// TIA Portal V15.1 export
// export: Created 2026-01-09T13:45:15.2149014Z, ExportSetting WithDefaults, WithReadOnly, DisplayName Totally Integrated Automation Portal, DisplayVersion V15.1 Update 8, DisplayName TIA Portal Openness, DisplayVersion V15.1 Update 8, DisplayName STEP 7 Professional, DisplayVersion V15.1 Update 8, DisplayName WinCC Advanced, DisplayVersion V15.1 Update 8
FUNCTION "FCCA_CCD_AGG12345" : Void   // FC19, LAD
{ S7_Optimized_Access := 'TRUE' }
VERSION : 0.1
// stored: AutoNumber true, CodeModifiedDate 2026-01-04T14:27:04.5188811Z, CompileDate 2026-01-04T14:27:06.4720109Z, CreationDate 2024-10-13T15:07:34.9617085Z, HandleErrorsWithinBlock false, InterfaceModifiedDate 2024-08-08T03:15:59.3806622Z, IsConsistent true, IsIECCheckEnabled false, IsKnowHowProtected false, IsWriteProtected false, LibraryConformanceStatus Error: The block contains calls of single instances. Warning: The object contains access to global data blocks. Warning: The block contains direct access to inputs, outputs, bit memories, indirect access to the registry or indirect access to external memory areas that are unknown at the time of compilation., ModifiedDate 2026-01-04T14:27:04.5188811Z, ParameterModified 2024-08-08T03:15:59.3806622Z, PLCSimAdvancedSupport false, SetENOAutomatically False, StructureModified 2024-08-08T03:15:59.3806622Z, UDAEnableTagReadback false
   VAR_TEMP   // added for the SCL form of the ladder/FBD networks
      _w1 : Bool;
   END_VAR
BEGIN

REGION Network 1: CAN COT LIEU AGG1
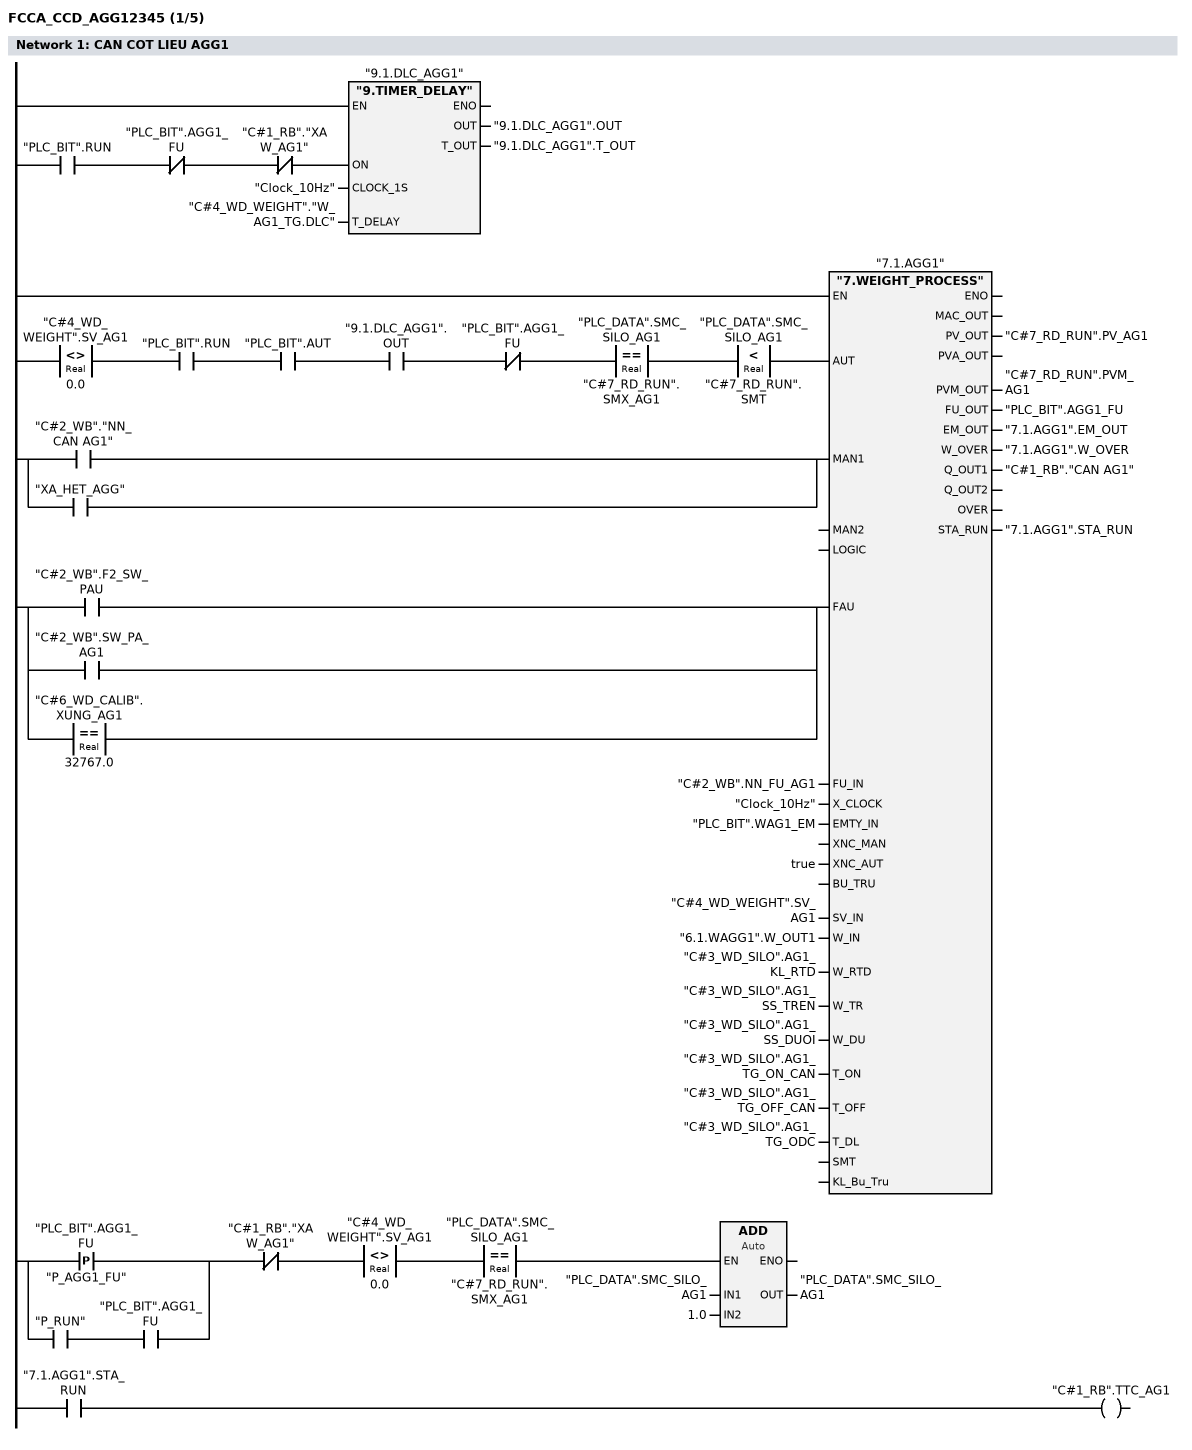
   RUNG wire#powerrail
      "9.1.DLC_AGG1"(ON := wire#w1, CLOCK_1S := "Clock_10Hz", T_DELAY := "C#4_WD_WEIGHT"."W_AG1_TG.DLC", OUT => "9.1.DLC_AGG1".OUT, T_OUT => "9.1.DLC_AGG1".T_OUT)
   END_RUNG
   RUNG wire#powerrail
      Contact( "PLC_BIT".RUN )
      I_Contact( "PLC_BIT".AGG1_FU )
      I_Contact( "C#1_RB"."XA W_AG1" )
   END_RUNG wire#w1
   RUNG wire#powerrail
      "7.1.AGG1"(AUT := wire#w2, MAN1 := wire#w3, FAU := wire#w4, MAN2 :=, LOGIC :=, FU_IN := "C#2_WB".NN_FU_AG1, X_CLOCK := "Clock_10Hz", EMTY_IN := "PLC_BIT".WAG1_EM, XNC_MAN :=, XNC_AUT := true, BU_TRU :=, SV_IN := "C#4_WD_WEIGHT".SV_AG1, W_IN := "6.1.WAGG1".W_OUT1, W_RTD := "C#3_WD_SILO".AG1_KL_RTD, W_TR := "C#3_WD_SILO".AG1_SS_TREN, W_DU := "C#3_WD_SILO".AG1_SS_DUOI, T_ON := "C#3_WD_SILO".AG1_TG_ON_CAN, T_OFF := "C#3_WD_SILO".AG1_TG_OFF_CAN, T_DL := "C#3_WD_SILO".AG1_TG_ODC, SMT :=, KL_Bu_Tru :=, MAC_OUT =>, PV_OUT => "C#7_RD_RUN".PV_AG1, PVA_OUT =>, PVM_OUT => "C#7_RD_RUN".PVM_AG1, FU_OUT => "PLC_BIT".AGG1_FU, EM_OUT => "7.1.AGG1".EM_OUT, W_OVER => "7.1.AGG1".W_OVER, Q_OUT1 => "C#1_RB"."CAN AG1", Q_OUT2 =>, OVER =>, STA_RUN => "7.1.AGG1".STA_RUN)
   END_RUNG
   RUNG wire#powerrail
      { S7_Templates := "SrcType := Real" } NE_Contact(in1 := "C#4_WD_WEIGHT".SV_AG1, in2 := 0.0)
      Contact( "PLC_BIT".RUN )
      Contact( "PLC_BIT".AUT )
      Contact( "9.1.DLC_AGG1".OUT )
      I_Contact( "PLC_BIT".AGG1_FU )
      { S7_Templates := "SrcType := Real" } EQ_Contact(in1 := "PLC_DATA".SMC_SILO_AG1, in2 := "C#7_RD_RUN".SMX_AG1)
      { S7_Templates := "SrcType := Real" } LT_Contact(in1 := "PLC_DATA".SMC_SILO_AG1, in2 := "C#7_RD_RUN".SMT)
   END_RUNG wire#w2
   RUNG wire#powerrail
      Contact( "C#2_WB"."NN_CAN AG1" )
   END_RUNG wire#w3
   RUNG wire#powerrail
      Contact( "XA_HET_AGG" )
   END_RUNG wire#w3
   RUNG wire#powerrail
      Contact( "C#2_WB".F2_SW_PAU )
   END_RUNG wire#w4
   RUNG wire#powerrail
      Contact( "C#2_WB".SW_PA_AG1 )
   END_RUNG wire#w4
   RUNG wire#powerrail
      { S7_Templates := "SrcType := Real" } EQ_Contact(in1 := "C#6_WD_CALIB".XUNG_AG1, in2 := 32767.0)
   END_RUNG wire#w4
   RUNG wire#powerrail
      P_Contact(operand := "PLC_BIT".AGG1_FU, bit := "P_AGG1_FU")
      wire#w5
      I_Contact( "C#1_RB"."XA W_AG1" )
      { S7_Templates := "SrcType := Real" } NE_Contact(in1 := "C#4_WD_WEIGHT".SV_AG1, in2 := 0.0)
      { S7_Templates := "SrcType := Real" } EQ_Contact(in1 := "PLC_DATA".SMC_SILO_AG1, in2 := "C#7_RD_RUN".SMX_AG1)
      Add(in1 := "PLC_DATA".SMC_SILO_AG1, in2 := 1.0, out => "PLC_DATA".SMC_SILO_AG1)
   END_RUNG
   RUNG wire#powerrail
      Contact( "P_RUN" )
      Contact( "PLC_BIT".AGG1_FU )
   END_RUNG wire#w5
   RUNG wire#powerrail
      Contact( "7.1.AGG1".STA_RUN )
      Coil( "C#1_RB".TTC_AG1 )
   END_RUNG
   // the same network as SCL:
   "9.1.DLC_AGG1"(ON := "PLC_BIT".RUN AND NOT "PLC_BIT".AGG1_FU AND NOT "C#1_RB"."XA W_AG1",   // "9.TIMER_DELAY"
                  CLOCK_1S := "Clock_10Hz",
                  T_DELAY := "C#4_WD_WEIGHT"."W_AG1_TG.DLC",
                  OUT => "9.1.DLC_AGG1".OUT,
                  T_OUT => "9.1.DLC_AGG1".T_OUT);
   "7.1.AGG1"(AUT := ("C#4_WD_WEIGHT".SV_AG1 <> 0.0) AND "PLC_BIT".RUN AND "PLC_BIT".AUT AND "9.1.DLC_AGG1".OUT AND NOT "PLC_BIT".AGG1_FU AND ("PLC_DATA".SMC_SILO_AG1 = "C#7_RD_RUN".SMX_AG1) AND ("PLC_DATA".SMC_SILO_AG1 < "C#7_RD_RUN".SMT),   // "7.WEIGHT_PROCESS"
              MAN1 := "C#2_WB"."NN_CAN AG1" OR "XA_HET_AGG",
              FAU := "C#2_WB".F2_SW_PAU OR "C#2_WB".SW_PA_AG1 OR ("C#6_WD_CALIB".XUNG_AG1 = 32767.0),
              FU_IN := "C#2_WB".NN_FU_AG1,
              X_CLOCK := "Clock_10Hz",
              EMTY_IN := "PLC_BIT".WAG1_EM,
              XNC_AUT := true,
              SV_IN := "C#4_WD_WEIGHT".SV_AG1,
              W_IN := "6.1.WAGG1".W_OUT1,
              W_RTD := "C#3_WD_SILO".AG1_KL_RTD,
              W_TR := "C#3_WD_SILO".AG1_SS_TREN,
              W_DU := "C#3_WD_SILO".AG1_SS_DUOI,
              T_ON := "C#3_WD_SILO".AG1_TG_ON_CAN,
              T_OFF := "C#3_WD_SILO".AG1_TG_OFF_CAN,
              T_DL := "C#3_WD_SILO".AG1_TG_ODC,
              PV_OUT => "C#7_RD_RUN".PV_AG1,
              PVM_OUT => "C#7_RD_RUN".PVM_AG1,
              FU_OUT => "PLC_BIT".AGG1_FU,
              EM_OUT => "7.1.AGG1".EM_OUT,
              W_OVER => "7.1.AGG1".W_OVER,
              Q_OUT1 => "C#1_RB"."CAN AG1",
              STA_RUN => "7.1.AGG1".STA_RUN);
   #_w1 := "PLC_BIT".AGG1_FU AND NOT "P_AGG1_FU";   // rising edge of "PLC_BIT".AGG1_FU
   "P_AGG1_FU" := "PLC_BIT".AGG1_FU;
   IF (#_w1 OR ("P_RUN" AND "PLC_BIT".AGG1_FU)) AND NOT "C#1_RB"."XA W_AG1" AND ("C#4_WD_WEIGHT".SV_AG1 <> 0.0) AND ("PLC_DATA".SMC_SILO_AG1 = "C#7_RD_RUN".SMX_AG1) THEN
       "PLC_DATA".SMC_SILO_AG1 := "PLC_DATA".SMC_SILO_AG1 + 1.0;
   END_IF;
   "C#1_RB".TTC_AG1 := "7.1.AGG1".STA_RUN;
END_REGION

REGION Network 2: CAN COT LIEU AGG2
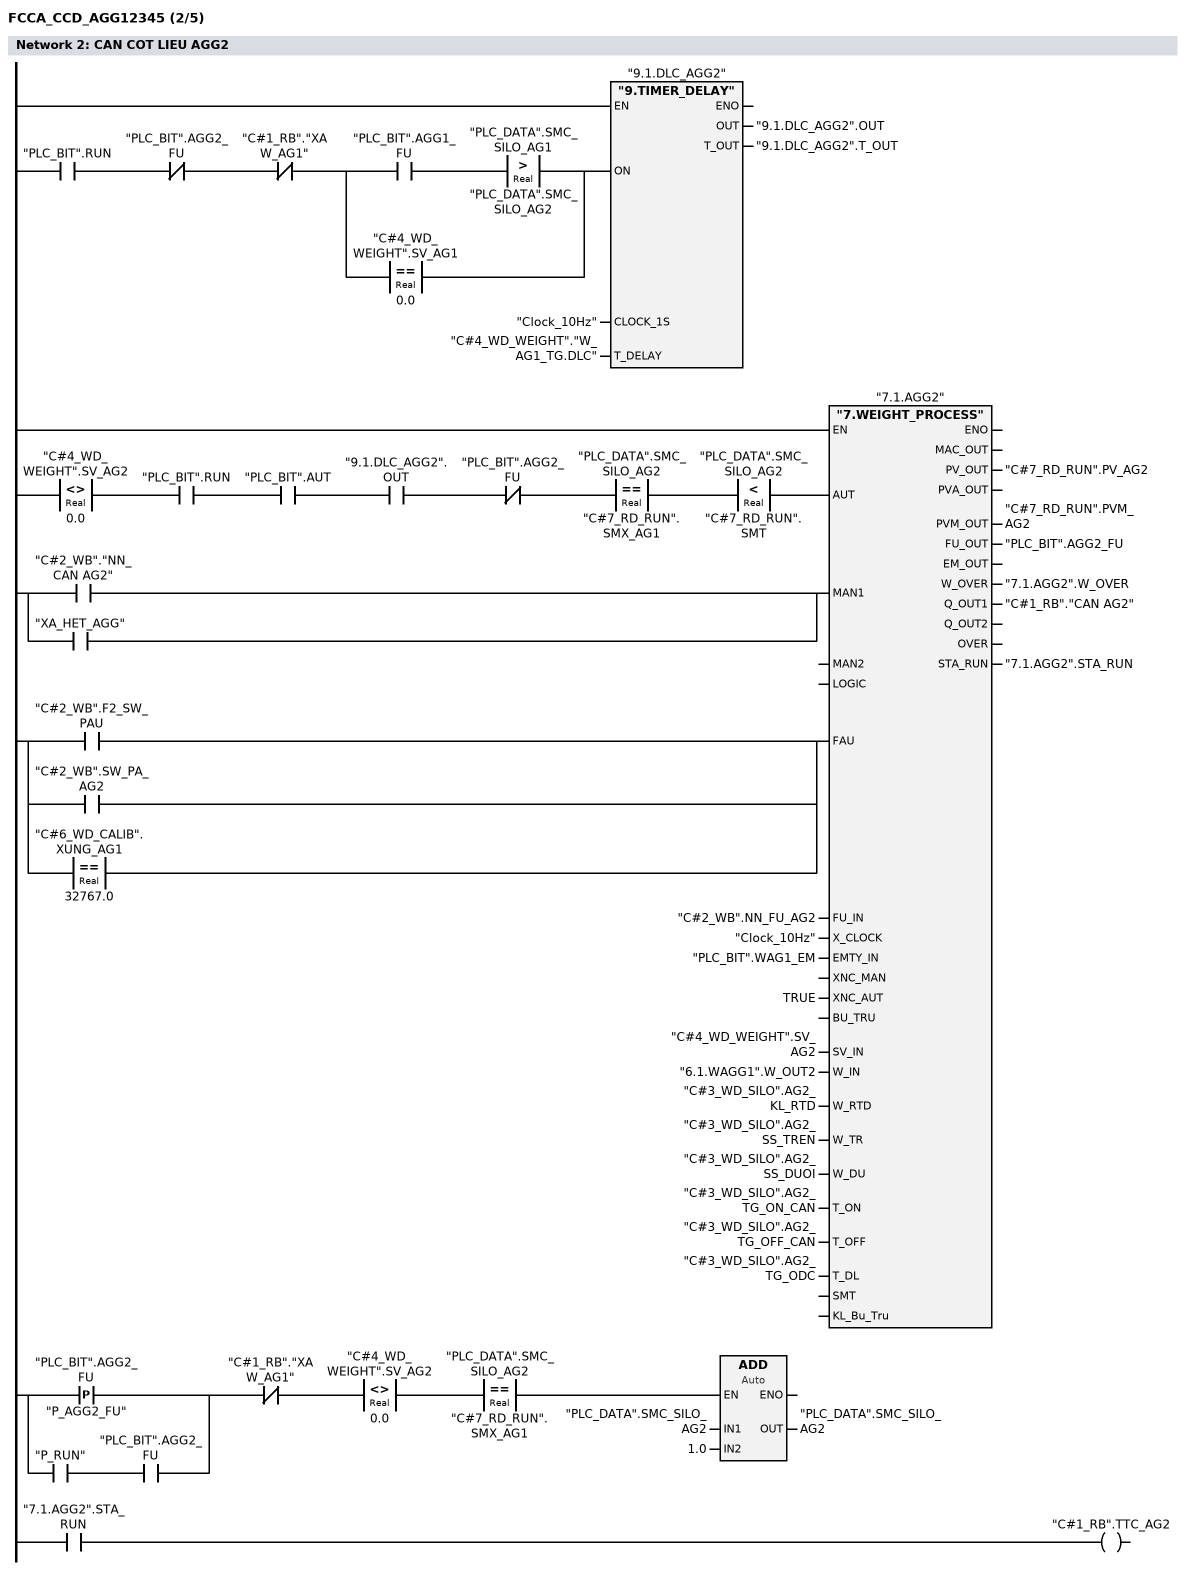
   RUNG wire#powerrail
      "9.1.DLC_AGG2"(ON := wire#w2, CLOCK_1S := "Clock_10Hz", T_DELAY := "C#4_WD_WEIGHT"."W_AG1_TG.DLC", OUT => "9.1.DLC_AGG2".OUT, T_OUT => "9.1.DLC_AGG2".T_OUT)
   END_RUNG
   RUNG wire#powerrail
      Contact( "PLC_BIT".RUN )
      I_Contact( "PLC_BIT".AGG2_FU )
      I_Contact( "C#1_RB"."XA W_AG1" )
      wire#w1
      Contact( "PLC_BIT".AGG1_FU )
      { S7_Templates := "SrcType := Real" } GT_Contact(in1 := "PLC_DATA".SMC_SILO_AG1, in2 := "PLC_DATA".SMC_SILO_AG2)
   END_RUNG wire#w2
   RUNG wire#w1
      { S7_Templates := "SrcType := Real" } EQ_Contact(in1 := "C#4_WD_WEIGHT".SV_AG1, in2 := 0.0)
   END_RUNG wire#w2
   RUNG wire#powerrail
      "7.1.AGG2"(AUT := wire#w3, MAN1 := wire#w4, FAU := wire#w5, MAN2 :=, LOGIC :=, FU_IN := "C#2_WB".NN_FU_AG2, X_CLOCK := "Clock_10Hz", EMTY_IN := "PLC_BIT".WAG1_EM, XNC_MAN :=, XNC_AUT := TRUE, BU_TRU :=, SV_IN := "C#4_WD_WEIGHT".SV_AG2, W_IN := "6.1.WAGG1".W_OUT2, W_RTD := "C#3_WD_SILO".AG2_KL_RTD, W_TR := "C#3_WD_SILO".AG2_SS_TREN, W_DU := "C#3_WD_SILO".AG2_SS_DUOI, T_ON := "C#3_WD_SILO".AG2_TG_ON_CAN, T_OFF := "C#3_WD_SILO".AG2_TG_OFF_CAN, T_DL := "C#3_WD_SILO".AG2_TG_ODC, SMT :=, KL_Bu_Tru :=, MAC_OUT =>, PV_OUT => "C#7_RD_RUN".PV_AG2, PVA_OUT =>, PVM_OUT => "C#7_RD_RUN".PVM_AG2, FU_OUT => "PLC_BIT".AGG2_FU, EM_OUT =>, W_OVER => "7.1.AGG2".W_OVER, Q_OUT1 => "C#1_RB"."CAN AG2", Q_OUT2 =>, OVER =>, STA_RUN => "7.1.AGG2".STA_RUN)
   END_RUNG
   RUNG wire#powerrail
      { S7_Templates := "SrcType := Real" } NE_Contact(in1 := "C#4_WD_WEIGHT".SV_AG2, in2 := 0.0)
      Contact( "PLC_BIT".RUN )
      Contact( "PLC_BIT".AUT )
      Contact( "9.1.DLC_AGG2".OUT )
      I_Contact( "PLC_BIT".AGG2_FU )
      { S7_Templates := "SrcType := Real" } EQ_Contact(in1 := "PLC_DATA".SMC_SILO_AG2, in2 := "C#7_RD_RUN".SMX_AG1)
      { S7_Templates := "SrcType := Real" } LT_Contact(in1 := "PLC_DATA".SMC_SILO_AG2, in2 := "C#7_RD_RUN".SMT)
   END_RUNG wire#w3
   RUNG wire#powerrail
      Contact( "C#2_WB"."NN_CAN AG2" )
   END_RUNG wire#w4
   RUNG wire#powerrail
      Contact( "XA_HET_AGG" )
   END_RUNG wire#w4
   RUNG wire#powerrail
      Contact( "C#2_WB".F2_SW_PAU )
   END_RUNG wire#w5
   RUNG wire#powerrail
      Contact( "C#2_WB".SW_PA_AG2 )
   END_RUNG wire#w5
   RUNG wire#powerrail
      { S7_Templates := "SrcType := Real" } EQ_Contact(in1 := "C#6_WD_CALIB".XUNG_AG1, in2 := 32767.0)
   END_RUNG wire#w5
   RUNG wire#powerrail
      P_Contact(operand := "PLC_BIT".AGG2_FU, bit := "P_AGG2_FU")
      wire#w6
      I_Contact( "C#1_RB"."XA W_AG1" )
      { S7_Templates := "SrcType := Real" } NE_Contact(in1 := "C#4_WD_WEIGHT".SV_AG2, in2 := 0.0)
      { S7_Templates := "SrcType := Real" } EQ_Contact(in1 := "PLC_DATA".SMC_SILO_AG2, in2 := "C#7_RD_RUN".SMX_AG1)
      Add(in1 := "PLC_DATA".SMC_SILO_AG2, in2 := 1.0, out => "PLC_DATA".SMC_SILO_AG2)
   END_RUNG
   RUNG wire#powerrail
      Contact( "P_RUN" )
      Contact( "PLC_BIT".AGG2_FU )
   END_RUNG wire#w6
   RUNG wire#powerrail
      Contact( "7.1.AGG2".STA_RUN )
      Coil( "C#1_RB".TTC_AG2 )
   END_RUNG
   // the same network as SCL:
   "9.1.DLC_AGG2"(ON := "PLC_BIT".RUN AND NOT "PLC_BIT".AGG2_FU AND NOT "C#1_RB"."XA W_AG1" AND (("PLC_BIT".AGG1_FU AND ("PLC_DATA".SMC_SILO_AG1 > "PLC_DATA".SMC_SILO_AG2)) OR ("C#4_WD_WEIGHT".SV_AG1 = 0.0)),   // "9.TIMER_DELAY"
                  CLOCK_1S := "Clock_10Hz",
                  T_DELAY := "C#4_WD_WEIGHT"."W_AG1_TG.DLC",
                  OUT => "9.1.DLC_AGG2".OUT,
                  T_OUT => "9.1.DLC_AGG2".T_OUT);
   "7.1.AGG2"(AUT := ("C#4_WD_WEIGHT".SV_AG2 <> 0.0) AND "PLC_BIT".RUN AND "PLC_BIT".AUT AND "9.1.DLC_AGG2".OUT AND NOT "PLC_BIT".AGG2_FU AND ("PLC_DATA".SMC_SILO_AG2 = "C#7_RD_RUN".SMX_AG1) AND ("PLC_DATA".SMC_SILO_AG2 < "C#7_RD_RUN".SMT),   // "7.WEIGHT_PROCESS"
              MAN1 := "C#2_WB"."NN_CAN AG2" OR "XA_HET_AGG",
              FAU := "C#2_WB".F2_SW_PAU OR "C#2_WB".SW_PA_AG2 OR ("C#6_WD_CALIB".XUNG_AG1 = 32767.0),
              FU_IN := "C#2_WB".NN_FU_AG2,
              X_CLOCK := "Clock_10Hz",
              EMTY_IN := "PLC_BIT".WAG1_EM,
              XNC_AUT := TRUE,
              SV_IN := "C#4_WD_WEIGHT".SV_AG2,
              W_IN := "6.1.WAGG1".W_OUT2,
              W_RTD := "C#3_WD_SILO".AG2_KL_RTD,
              W_TR := "C#3_WD_SILO".AG2_SS_TREN,
              W_DU := "C#3_WD_SILO".AG2_SS_DUOI,
              T_ON := "C#3_WD_SILO".AG2_TG_ON_CAN,
              T_OFF := "C#3_WD_SILO".AG2_TG_OFF_CAN,
              T_DL := "C#3_WD_SILO".AG2_TG_ODC,
              PV_OUT => "C#7_RD_RUN".PV_AG2,
              PVM_OUT => "C#7_RD_RUN".PVM_AG2,
              FU_OUT => "PLC_BIT".AGG2_FU,
              W_OVER => "7.1.AGG2".W_OVER,
              Q_OUT1 => "C#1_RB"."CAN AG2",
              STA_RUN => "7.1.AGG2".STA_RUN);
   #_w1 := "PLC_BIT".AGG2_FU AND NOT "P_AGG2_FU";   // rising edge of "PLC_BIT".AGG2_FU
   "P_AGG2_FU" := "PLC_BIT".AGG2_FU;
   IF (#_w1 OR ("P_RUN" AND "PLC_BIT".AGG2_FU)) AND NOT "C#1_RB"."XA W_AG1" AND ("C#4_WD_WEIGHT".SV_AG2 <> 0.0) AND ("PLC_DATA".SMC_SILO_AG2 = "C#7_RD_RUN".SMX_AG1) THEN
       "PLC_DATA".SMC_SILO_AG2 := "PLC_DATA".SMC_SILO_AG2 + 1.0;
   END_IF;
   "C#1_RB".TTC_AG2 := "7.1.AGG2".STA_RUN;
END_REGION

REGION Network 3: CAN COT LIEU AGG3
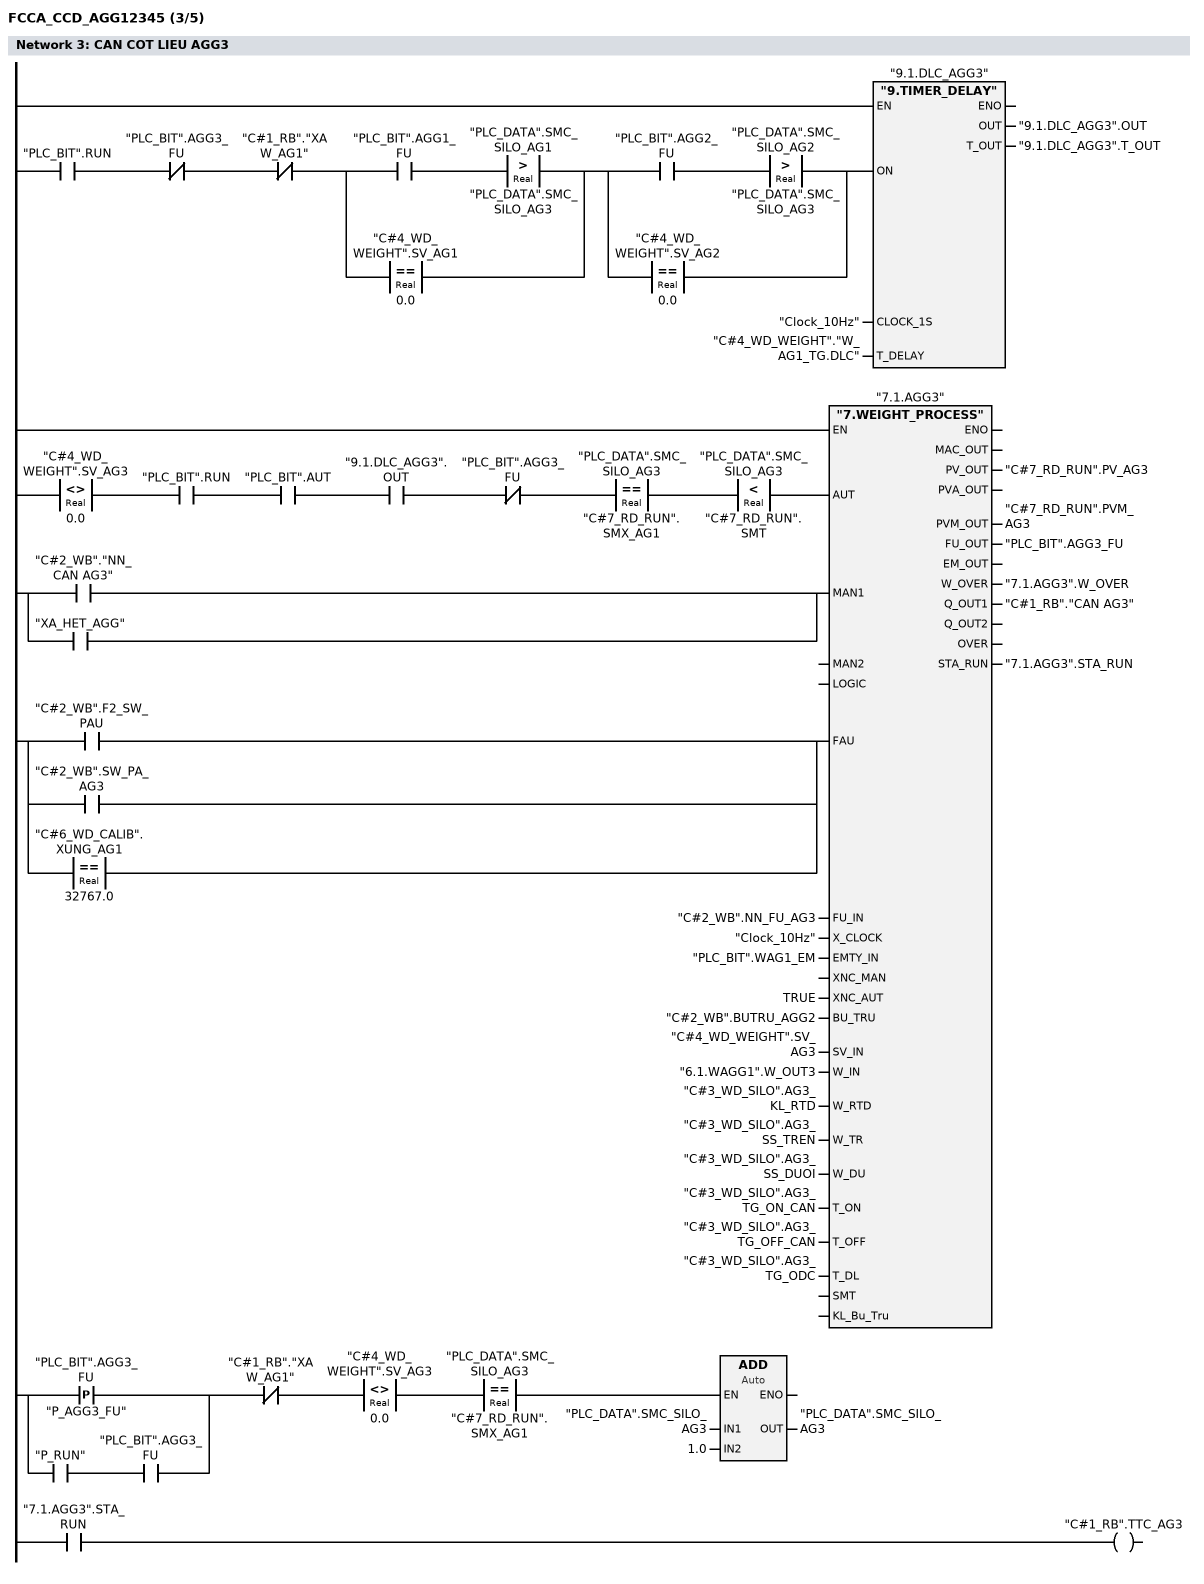
   RUNG wire#powerrail
      "9.1.DLC_AGG3"(ON := wire#w3, CLOCK_1S := "Clock_10Hz", T_DELAY := "C#4_WD_WEIGHT"."W_AG1_TG.DLC", OUT => "9.1.DLC_AGG3".OUT, T_OUT => "9.1.DLC_AGG3".T_OUT)
   END_RUNG
   RUNG wire#powerrail
      Contact( "PLC_BIT".RUN )
      I_Contact( "PLC_BIT".AGG3_FU )
      I_Contact( "C#1_RB"."XA W_AG1" )
      wire#w1
      Contact( "PLC_BIT".AGG1_FU )
      { S7_Templates := "SrcType := Real" } GT_Contact(in1 := "PLC_DATA".SMC_SILO_AG1, in2 := "PLC_DATA".SMC_SILO_AG3)
      wire#w2
      Contact( "PLC_BIT".AGG2_FU )
      { S7_Templates := "SrcType := Real" } GT_Contact(in1 := "PLC_DATA".SMC_SILO_AG2, in2 := "PLC_DATA".SMC_SILO_AG3)
   END_RUNG wire#w3
   RUNG wire#w1
      { S7_Templates := "SrcType := Real" } EQ_Contact(in1 := "C#4_WD_WEIGHT".SV_AG1, in2 := 0.0)
   END_RUNG wire#w2
   RUNG wire#w2
      { S7_Templates := "SrcType := Real" } EQ_Contact(in1 := "C#4_WD_WEIGHT".SV_AG2, in2 := 0.0)
   END_RUNG wire#w3
   RUNG wire#powerrail
      "7.1.AGG3"(AUT := wire#w4, MAN1 := wire#w5, FAU := wire#w6, MAN2 :=, LOGIC :=, FU_IN := "C#2_WB".NN_FU_AG3, X_CLOCK := "Clock_10Hz", EMTY_IN := "PLC_BIT".WAG1_EM, XNC_MAN :=, XNC_AUT := TRUE, BU_TRU := "C#2_WB".BUTRU_AGG2, SV_IN := "C#4_WD_WEIGHT".SV_AG3, W_IN := "6.1.WAGG1".W_OUT3, W_RTD := "C#3_WD_SILO".AG3_KL_RTD, W_TR := "C#3_WD_SILO".AG3_SS_TREN, W_DU := "C#3_WD_SILO".AG3_SS_DUOI, T_ON := "C#3_WD_SILO".AG3_TG_ON_CAN, T_OFF := "C#3_WD_SILO".AG3_TG_OFF_CAN, T_DL := "C#3_WD_SILO".AG3_TG_ODC, SMT :=, KL_Bu_Tru :=, MAC_OUT =>, PV_OUT => "C#7_RD_RUN".PV_AG3, PVA_OUT =>, PVM_OUT => "C#7_RD_RUN".PVM_AG3, FU_OUT => "PLC_BIT".AGG3_FU, EM_OUT =>, W_OVER => "7.1.AGG3".W_OVER, Q_OUT1 => "C#1_RB"."CAN AG3", Q_OUT2 =>, OVER =>, STA_RUN => "7.1.AGG3".STA_RUN)
   END_RUNG
   RUNG wire#powerrail
      { S7_Templates := "SrcType := Real" } NE_Contact(in1 := "C#4_WD_WEIGHT".SV_AG3, in2 := 0.0)
      Contact( "PLC_BIT".RUN )
      Contact( "PLC_BIT".AUT )
      Contact( "9.1.DLC_AGG3".OUT )
      I_Contact( "PLC_BIT".AGG3_FU )
      { S7_Templates := "SrcType := Real" } EQ_Contact(in1 := "PLC_DATA".SMC_SILO_AG3, in2 := "C#7_RD_RUN".SMX_AG1)
      { S7_Templates := "SrcType := Real" } LT_Contact(in1 := "PLC_DATA".SMC_SILO_AG3, in2 := "C#7_RD_RUN".SMT)
   END_RUNG wire#w4
   RUNG wire#powerrail
      Contact( "C#2_WB"."NN_CAN AG3" )
   END_RUNG wire#w5
   RUNG wire#powerrail
      Contact( "XA_HET_AGG" )
   END_RUNG wire#w5
   RUNG wire#powerrail
      Contact( "C#2_WB".F2_SW_PAU )
   END_RUNG wire#w6
   RUNG wire#powerrail
      Contact( "C#2_WB".SW_PA_AG3 )
   END_RUNG wire#w6
   RUNG wire#powerrail
      { S7_Templates := "SrcType := Real" } EQ_Contact(in1 := "C#6_WD_CALIB".XUNG_AG1, in2 := 32767.0)
   END_RUNG wire#w6
   RUNG wire#powerrail
      P_Contact(operand := "PLC_BIT".AGG3_FU, bit := "P_AGG3_FU")
      wire#w7
      I_Contact( "C#1_RB"."XA W_AG1" )
      { S7_Templates := "SrcType := Real" } NE_Contact(in1 := "C#4_WD_WEIGHT".SV_AG3, in2 := 0.0)
      { S7_Templates := "SrcType := Real" } EQ_Contact(in1 := "PLC_DATA".SMC_SILO_AG3, in2 := "C#7_RD_RUN".SMX_AG1)
      Add(in1 := "PLC_DATA".SMC_SILO_AG3, in2 := 1.0, out => "PLC_DATA".SMC_SILO_AG3)
   END_RUNG
   RUNG wire#powerrail
      Contact( "P_RUN" )
      Contact( "PLC_BIT".AGG3_FU )
   END_RUNG wire#w7
   RUNG wire#powerrail
      Contact( "7.1.AGG3".STA_RUN )
      Coil( "C#1_RB".TTC_AG3 )
   END_RUNG
   // the same network as SCL:
   "9.1.DLC_AGG3"(ON := "PLC_BIT".RUN AND NOT "PLC_BIT".AGG3_FU AND NOT "C#1_RB"."XA W_AG1" AND (("PLC_BIT".AGG1_FU AND ("PLC_DATA".SMC_SILO_AG1 > "PLC_DATA".SMC_SILO_AG3)) OR ("C#4_WD_WEIGHT".SV_AG1 = 0.0)) AND (("PLC_BIT".AGG2_FU AND ("PLC_DATA".SMC_SILO_AG2 > "PLC_DATA".SMC_SILO_AG3)) OR ("C#4_WD_WEIGHT".SV_AG2 = 0.0)),   // "9.TIMER_DELAY"
                  CLOCK_1S := "Clock_10Hz",
                  T_DELAY := "C#4_WD_WEIGHT"."W_AG1_TG.DLC",
                  OUT => "9.1.DLC_AGG3".OUT,
                  T_OUT => "9.1.DLC_AGG3".T_OUT);
   "7.1.AGG3"(AUT := ("C#4_WD_WEIGHT".SV_AG3 <> 0.0) AND "PLC_BIT".RUN AND "PLC_BIT".AUT AND "9.1.DLC_AGG3".OUT AND NOT "PLC_BIT".AGG3_FU AND ("PLC_DATA".SMC_SILO_AG3 = "C#7_RD_RUN".SMX_AG1) AND ("PLC_DATA".SMC_SILO_AG3 < "C#7_RD_RUN".SMT),   // "7.WEIGHT_PROCESS"
              MAN1 := "C#2_WB"."NN_CAN AG3" OR "XA_HET_AGG",
              FAU := "C#2_WB".F2_SW_PAU OR "C#2_WB".SW_PA_AG3 OR ("C#6_WD_CALIB".XUNG_AG1 = 32767.0),
              FU_IN := "C#2_WB".NN_FU_AG3,
              X_CLOCK := "Clock_10Hz",
              EMTY_IN := "PLC_BIT".WAG1_EM,
              XNC_AUT := TRUE,
              BU_TRU := "C#2_WB".BUTRU_AGG2,
              SV_IN := "C#4_WD_WEIGHT".SV_AG3,
              W_IN := "6.1.WAGG1".W_OUT3,
              W_RTD := "C#3_WD_SILO".AG3_KL_RTD,
              W_TR := "C#3_WD_SILO".AG3_SS_TREN,
              W_DU := "C#3_WD_SILO".AG3_SS_DUOI,
              T_ON := "C#3_WD_SILO".AG3_TG_ON_CAN,
              T_OFF := "C#3_WD_SILO".AG3_TG_OFF_CAN,
              T_DL := "C#3_WD_SILO".AG3_TG_ODC,
              PV_OUT => "C#7_RD_RUN".PV_AG3,
              PVM_OUT => "C#7_RD_RUN".PVM_AG3,
              FU_OUT => "PLC_BIT".AGG3_FU,
              W_OVER => "7.1.AGG3".W_OVER,
              Q_OUT1 => "C#1_RB"."CAN AG3",
              STA_RUN => "7.1.AGG3".STA_RUN);
   #_w1 := "PLC_BIT".AGG3_FU AND NOT "P_AGG3_FU";   // rising edge of "PLC_BIT".AGG3_FU
   "P_AGG3_FU" := "PLC_BIT".AGG3_FU;
   IF (#_w1 OR ("P_RUN" AND "PLC_BIT".AGG3_FU)) AND NOT "C#1_RB"."XA W_AG1" AND ("C#4_WD_WEIGHT".SV_AG3 <> 0.0) AND ("PLC_DATA".SMC_SILO_AG3 = "C#7_RD_RUN".SMX_AG1) THEN
       "PLC_DATA".SMC_SILO_AG3 := "PLC_DATA".SMC_SILO_AG3 + 1.0;
   END_IF;
   "C#1_RB".TTC_AG3 := "7.1.AGG3".STA_RUN;
END_REGION

REGION Network 4: CAN COT LIEU AGG4
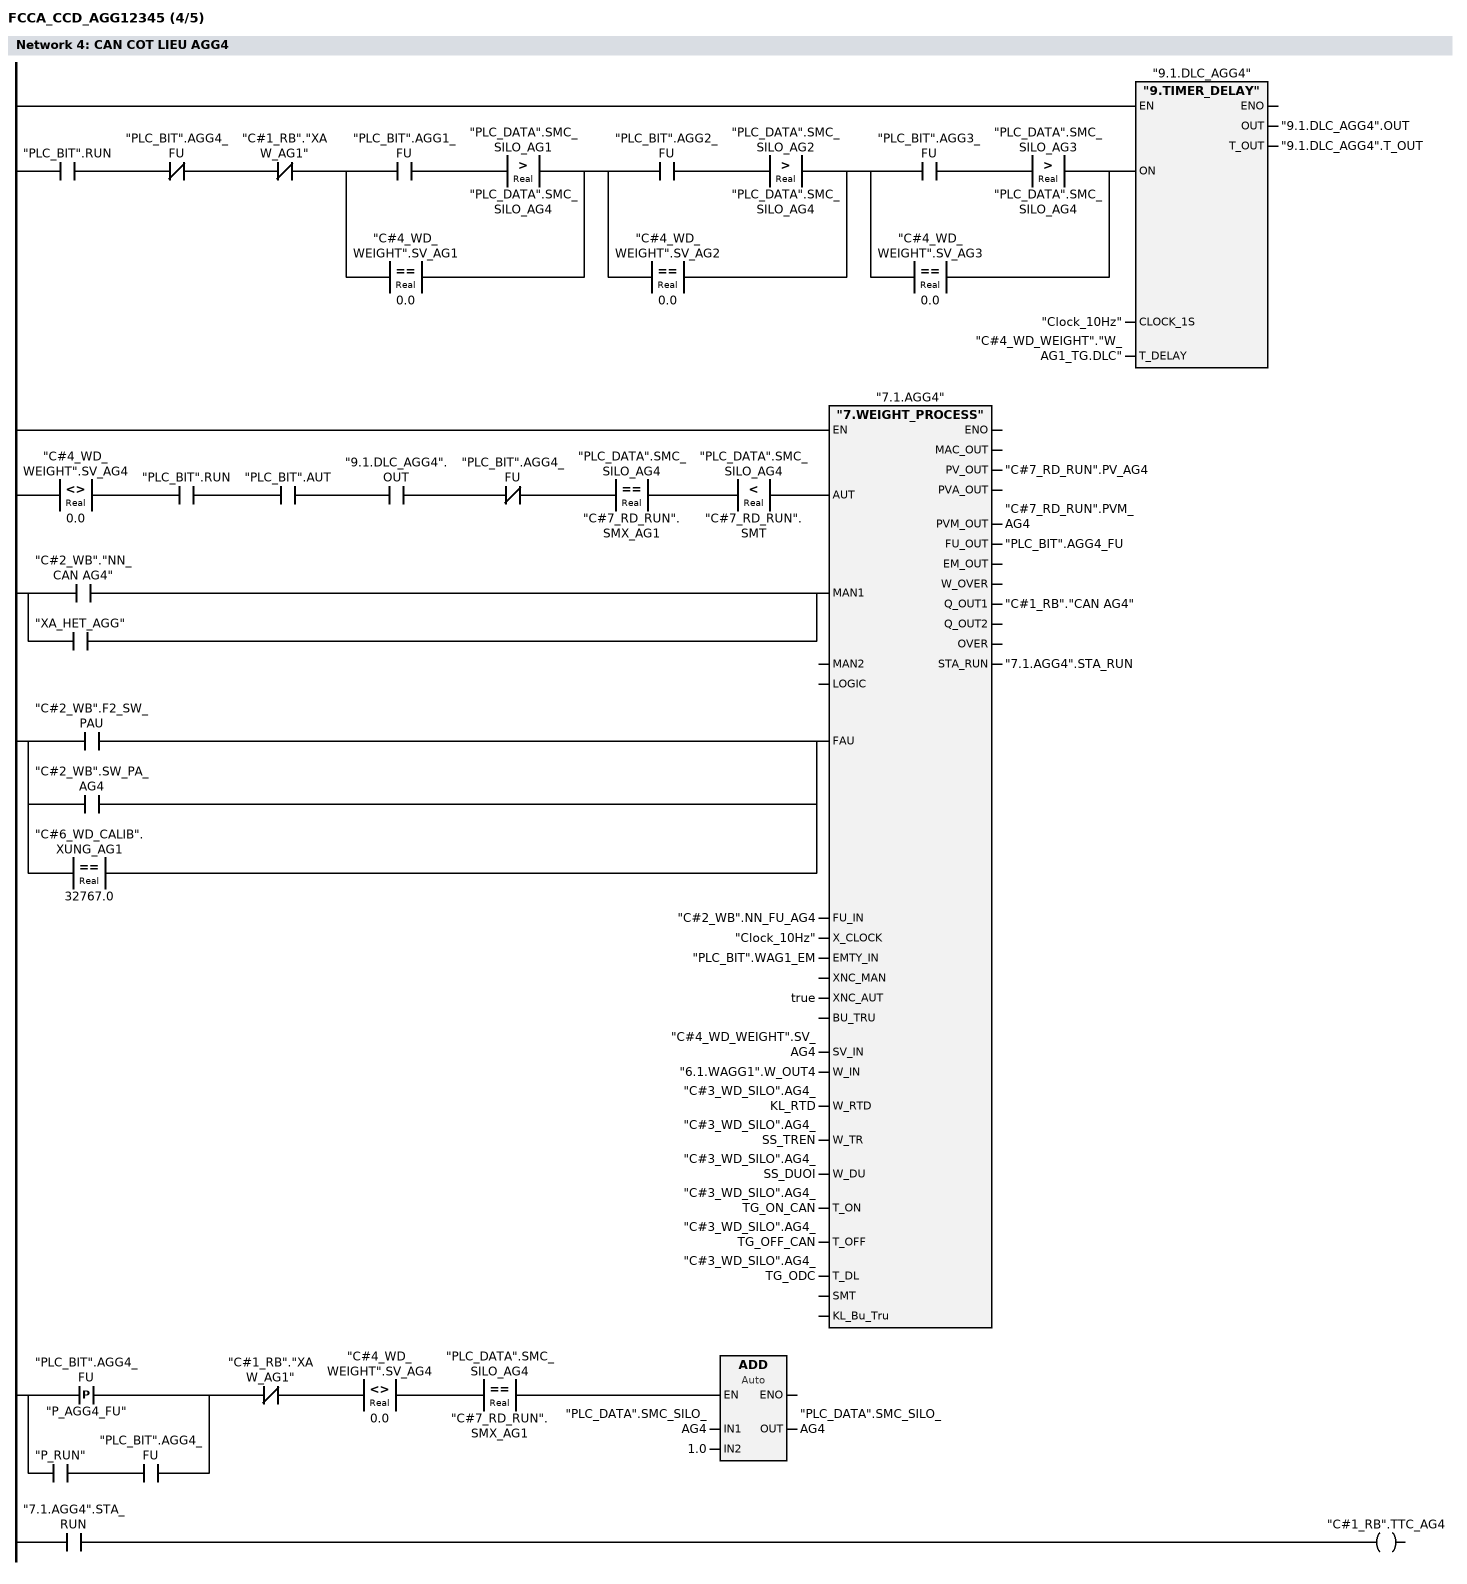
   RUNG wire#powerrail
      "9.1.DLC_AGG4"(ON := wire#w4, CLOCK_1S := "Clock_10Hz", T_DELAY := "C#4_WD_WEIGHT"."W_AG1_TG.DLC", OUT => "9.1.DLC_AGG4".OUT, T_OUT => "9.1.DLC_AGG4".T_OUT)
   END_RUNG
   RUNG wire#powerrail
      Contact( "PLC_BIT".RUN )
      I_Contact( "PLC_BIT".AGG4_FU )
      I_Contact( "C#1_RB"."XA W_AG1" )
      wire#w1
      Contact( "PLC_BIT".AGG1_FU )
      { S7_Templates := "SrcType := Real" } GT_Contact(in1 := "PLC_DATA".SMC_SILO_AG1, in2 := "PLC_DATA".SMC_SILO_AG4)
      wire#w2
      Contact( "PLC_BIT".AGG2_FU )
      { S7_Templates := "SrcType := Real" } GT_Contact(in1 := "PLC_DATA".SMC_SILO_AG2, in2 := "PLC_DATA".SMC_SILO_AG4)
      wire#w3
      Contact( "PLC_BIT".AGG3_FU )
      { S7_Templates := "SrcType := Real" } GT_Contact(in1 := "PLC_DATA".SMC_SILO_AG3, in2 := "PLC_DATA".SMC_SILO_AG4)
   END_RUNG wire#w4
   RUNG wire#w1
      { S7_Templates := "SrcType := Real" } EQ_Contact(in1 := "C#4_WD_WEIGHT".SV_AG1, in2 := 0.0)
   END_RUNG wire#w2
   RUNG wire#w2
      { S7_Templates := "SrcType := Real" } EQ_Contact(in1 := "C#4_WD_WEIGHT".SV_AG2, in2 := 0.0)
   END_RUNG wire#w3
   RUNG wire#w3
      { S7_Templates := "SrcType := Real" } EQ_Contact(in1 := "C#4_WD_WEIGHT".SV_AG3, in2 := 0.0)
   END_RUNG wire#w4
   RUNG wire#powerrail
      "7.1.AGG4"(AUT := wire#w5, MAN1 := wire#w6, FAU := wire#w7, MAN2 :=, LOGIC :=, FU_IN := "C#2_WB".NN_FU_AG4, X_CLOCK := "Clock_10Hz", EMTY_IN := "PLC_BIT".WAG1_EM, XNC_MAN :=, XNC_AUT := true, BU_TRU :=, SV_IN := "C#4_WD_WEIGHT".SV_AG4, W_IN := "6.1.WAGG1".W_OUT4, W_RTD := "C#3_WD_SILO".AG4_KL_RTD, W_TR := "C#3_WD_SILO".AG4_SS_TREN, W_DU := "C#3_WD_SILO".AG4_SS_DUOI, T_ON := "C#3_WD_SILO".AG4_TG_ON_CAN, T_OFF := "C#3_WD_SILO".AG4_TG_OFF_CAN, T_DL := "C#3_WD_SILO".AG4_TG_ODC, SMT :=, KL_Bu_Tru :=, MAC_OUT =>, PV_OUT => "C#7_RD_RUN".PV_AG4, PVA_OUT =>, PVM_OUT => "C#7_RD_RUN".PVM_AG4, FU_OUT => "PLC_BIT".AGG4_FU, EM_OUT =>, W_OVER =>, Q_OUT1 => "C#1_RB"."CAN AG4", Q_OUT2 =>, OVER =>, STA_RUN => "7.1.AGG4".STA_RUN)
   END_RUNG
   RUNG wire#powerrail
      { S7_Templates := "SrcType := Real" } NE_Contact(in1 := "C#4_WD_WEIGHT".SV_AG4, in2 := 0.0)
      Contact( "PLC_BIT".RUN )
      Contact( "PLC_BIT".AUT )
      Contact( "9.1.DLC_AGG4".OUT )
      I_Contact( "PLC_BIT".AGG4_FU )
      { S7_Templates := "SrcType := Real" } EQ_Contact(in1 := "PLC_DATA".SMC_SILO_AG4, in2 := "C#7_RD_RUN".SMX_AG1)
      { S7_Templates := "SrcType := Real" } LT_Contact(in1 := "PLC_DATA".SMC_SILO_AG4, in2 := "C#7_RD_RUN".SMT)
   END_RUNG wire#w5
   RUNG wire#powerrail
      Contact( "C#2_WB"."NN_CAN AG4" )
   END_RUNG wire#w6
   RUNG wire#powerrail
      Contact( "XA_HET_AGG" )
   END_RUNG wire#w6
   RUNG wire#powerrail
      Contact( "C#2_WB".F2_SW_PAU )
   END_RUNG wire#w7
   RUNG wire#powerrail
      Contact( "C#2_WB".SW_PA_AG4 )
   END_RUNG wire#w7
   RUNG wire#powerrail
      { S7_Templates := "SrcType := Real" } EQ_Contact(in1 := "C#6_WD_CALIB".XUNG_AG1, in2 := 32767.0)
   END_RUNG wire#w7
   RUNG wire#powerrail
      P_Contact(operand := "PLC_BIT".AGG4_FU, bit := "P_AGG4_FU")
      wire#w8
      I_Contact( "C#1_RB"."XA W_AG1" )
      { S7_Templates := "SrcType := Real" } NE_Contact(in1 := "C#4_WD_WEIGHT".SV_AG4, in2 := 0.0)
      { S7_Templates := "SrcType := Real" } EQ_Contact(in1 := "PLC_DATA".SMC_SILO_AG4, in2 := "C#7_RD_RUN".SMX_AG1)
      Add(in1 := "PLC_DATA".SMC_SILO_AG4, in2 := 1.0, out => "PLC_DATA".SMC_SILO_AG4)
   END_RUNG
   RUNG wire#powerrail
      Contact( "P_RUN" )
      Contact( "PLC_BIT".AGG4_FU )
   END_RUNG wire#w8
   RUNG wire#powerrail
      Contact( "7.1.AGG4".STA_RUN )
      Coil( "C#1_RB".TTC_AG4 )
   END_RUNG
   // the same network as SCL:
   "9.1.DLC_AGG4"(ON := "PLC_BIT".RUN AND NOT "PLC_BIT".AGG4_FU AND NOT "C#1_RB"."XA W_AG1" AND (("PLC_BIT".AGG1_FU AND ("PLC_DATA".SMC_SILO_AG1 > "PLC_DATA".SMC_SILO_AG4)) OR ("C#4_WD_WEIGHT".SV_AG1 = 0.0)) AND (("PLC_BIT".AGG2_FU AND ("PLC_DATA".SMC_SILO_AG2 > "PLC_DATA".SMC_SILO_AG4)) OR ("C#4_WD_WEIGHT".SV_AG2 = 0.0)) AND (("PLC_BIT".AGG3_FU AND ("PLC_DATA".SMC_SILO_AG3 > "PLC_DATA".SMC_SILO_AG4)) OR ("C#4_WD_WEIGHT".SV_AG3 = 0.0)),   // "9.TIMER_DELAY"
                  CLOCK_1S := "Clock_10Hz",
                  T_DELAY := "C#4_WD_WEIGHT"."W_AG1_TG.DLC",
                  OUT => "9.1.DLC_AGG4".OUT,
                  T_OUT => "9.1.DLC_AGG4".T_OUT);
   "7.1.AGG4"(AUT := ("C#4_WD_WEIGHT".SV_AG4 <> 0.0) AND "PLC_BIT".RUN AND "PLC_BIT".AUT AND "9.1.DLC_AGG4".OUT AND NOT "PLC_BIT".AGG4_FU AND ("PLC_DATA".SMC_SILO_AG4 = "C#7_RD_RUN".SMX_AG1) AND ("PLC_DATA".SMC_SILO_AG4 < "C#7_RD_RUN".SMT),   // "7.WEIGHT_PROCESS"
              MAN1 := "C#2_WB"."NN_CAN AG4" OR "XA_HET_AGG",
              FAU := "C#2_WB".F2_SW_PAU OR "C#2_WB".SW_PA_AG4 OR ("C#6_WD_CALIB".XUNG_AG1 = 32767.0),
              FU_IN := "C#2_WB".NN_FU_AG4,
              X_CLOCK := "Clock_10Hz",
              EMTY_IN := "PLC_BIT".WAG1_EM,
              XNC_AUT := true,
              SV_IN := "C#4_WD_WEIGHT".SV_AG4,
              W_IN := "6.1.WAGG1".W_OUT4,
              W_RTD := "C#3_WD_SILO".AG4_KL_RTD,
              W_TR := "C#3_WD_SILO".AG4_SS_TREN,
              W_DU := "C#3_WD_SILO".AG4_SS_DUOI,
              T_ON := "C#3_WD_SILO".AG4_TG_ON_CAN,
              T_OFF := "C#3_WD_SILO".AG4_TG_OFF_CAN,
              T_DL := "C#3_WD_SILO".AG4_TG_ODC,
              PV_OUT => "C#7_RD_RUN".PV_AG4,
              PVM_OUT => "C#7_RD_RUN".PVM_AG4,
              FU_OUT => "PLC_BIT".AGG4_FU,
              Q_OUT1 => "C#1_RB"."CAN AG4",
              STA_RUN => "7.1.AGG4".STA_RUN);
   #_w1 := "PLC_BIT".AGG4_FU AND NOT "P_AGG4_FU";   // rising edge of "PLC_BIT".AGG4_FU
   "P_AGG4_FU" := "PLC_BIT".AGG4_FU;
   IF (#_w1 OR ("P_RUN" AND "PLC_BIT".AGG4_FU)) AND NOT "C#1_RB"."XA W_AG1" AND ("C#4_WD_WEIGHT".SV_AG4 <> 0.0) AND ("PLC_DATA".SMC_SILO_AG4 = "C#7_RD_RUN".SMX_AG1) THEN
       "PLC_DATA".SMC_SILO_AG4 := "PLC_DATA".SMC_SILO_AG4 + 1.0;
   END_IF;
   "C#1_RB".TTC_AG4 := "7.1.AGG4".STA_RUN;
END_REGION

REGION Network 5: Trạng thái cân Ag4
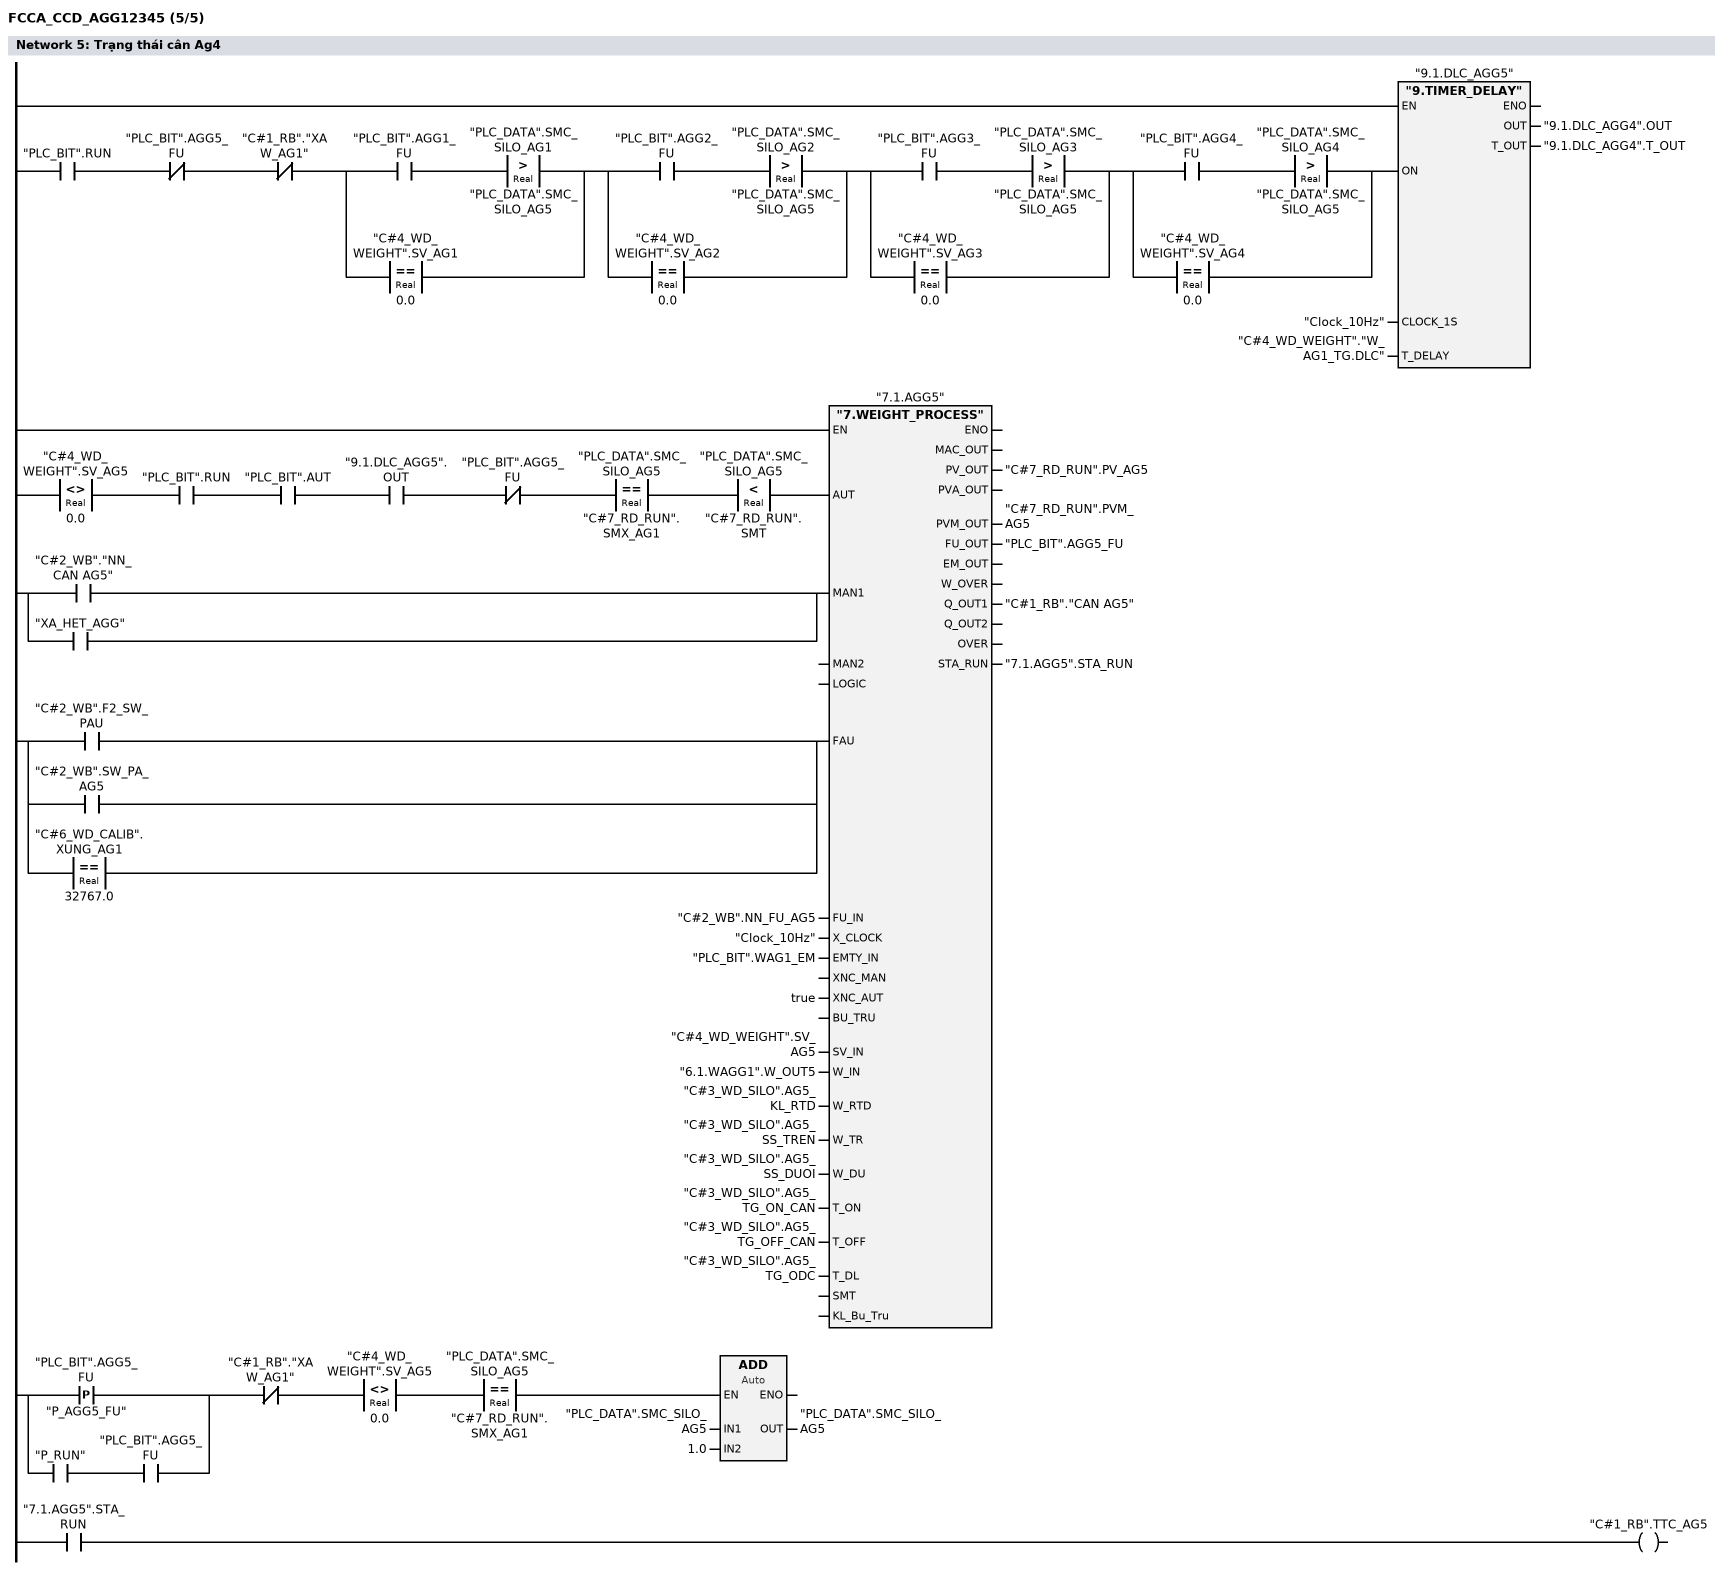
   RUNG wire#powerrail
      "9.1.DLC_AGG5"(ON := wire#w5, CLOCK_1S := "Clock_10Hz", T_DELAY := "C#4_WD_WEIGHT"."W_AG1_TG.DLC", OUT => "9.1.DLC_AGG4".OUT, T_OUT => "9.1.DLC_AGG4".T_OUT)
   END_RUNG
   RUNG wire#powerrail
      Contact( "PLC_BIT".RUN )
      I_Contact( "PLC_BIT".AGG5_FU )
      I_Contact( "C#1_RB"."XA W_AG1" )
      wire#w1
      Contact( "PLC_BIT".AGG1_FU )
      { S7_Templates := "SrcType := Real" } GT_Contact(in1 := "PLC_DATA".SMC_SILO_AG1, in2 := "PLC_DATA".SMC_SILO_AG5)
      wire#w2
      Contact( "PLC_BIT".AGG2_FU )
      { S7_Templates := "SrcType := Real" } GT_Contact(in1 := "PLC_DATA".SMC_SILO_AG2, in2 := "PLC_DATA".SMC_SILO_AG5)
      wire#w3
      Contact( "PLC_BIT".AGG3_FU )
      { S7_Templates := "SrcType := Real" } GT_Contact(in1 := "PLC_DATA".SMC_SILO_AG3, in2 := "PLC_DATA".SMC_SILO_AG5)
      wire#w4
      Contact( "PLC_BIT".AGG4_FU )
      { S7_Templates := "SrcType := Real" } GT_Contact(in1 := "PLC_DATA".SMC_SILO_AG4, in2 := "PLC_DATA".SMC_SILO_AG5)
   END_RUNG wire#w5
   RUNG wire#w1
      { S7_Templates := "SrcType := Real" } EQ_Contact(in1 := "C#4_WD_WEIGHT".SV_AG1, in2 := 0.0)
   END_RUNG wire#w2
   RUNG wire#w2
      { S7_Templates := "SrcType := Real" } EQ_Contact(in1 := "C#4_WD_WEIGHT".SV_AG2, in2 := 0.0)
   END_RUNG wire#w3
   RUNG wire#w3
      { S7_Templates := "SrcType := Real" } EQ_Contact(in1 := "C#4_WD_WEIGHT".SV_AG3, in2 := 0.0)
   END_RUNG wire#w4
   RUNG wire#w4
      { S7_Templates := "SrcType := Real" } EQ_Contact(in1 := "C#4_WD_WEIGHT".SV_AG4, in2 := 0.0)
   END_RUNG wire#w5
   RUNG wire#powerrail
      "7.1.AGG5"(AUT := wire#w6, MAN1 := wire#w7, FAU := wire#w8, MAN2 :=, LOGIC :=, FU_IN := "C#2_WB".NN_FU_AG5, X_CLOCK := "Clock_10Hz", EMTY_IN := "PLC_BIT".WAG1_EM, XNC_MAN :=, XNC_AUT := true, BU_TRU :=, SV_IN := "C#4_WD_WEIGHT".SV_AG5, W_IN := "6.1.WAGG1".W_OUT5, W_RTD := "C#3_WD_SILO".AG5_KL_RTD, W_TR := "C#3_WD_SILO".AG5_SS_TREN, W_DU := "C#3_WD_SILO".AG5_SS_DUOI, T_ON := "C#3_WD_SILO".AG5_TG_ON_CAN, T_OFF := "C#3_WD_SILO".AG5_TG_OFF_CAN, T_DL := "C#3_WD_SILO".AG5_TG_ODC, SMT :=, KL_Bu_Tru :=, MAC_OUT =>, PV_OUT => "C#7_RD_RUN".PV_AG5, PVA_OUT =>, PVM_OUT => "C#7_RD_RUN".PVM_AG5, FU_OUT => "PLC_BIT".AGG5_FU, EM_OUT =>, W_OVER =>, Q_OUT1 => "C#1_RB"."CAN AG5", Q_OUT2 =>, OVER =>, STA_RUN => "7.1.AGG5".STA_RUN)
   END_RUNG
   RUNG wire#powerrail
      { S7_Templates := "SrcType := Real" } NE_Contact(in1 := "C#4_WD_WEIGHT".SV_AG5, in2 := 0.0)
      Contact( "PLC_BIT".RUN )
      Contact( "PLC_BIT".AUT )
      Contact( "9.1.DLC_AGG5".OUT )
      I_Contact( "PLC_BIT".AGG5_FU )
      { S7_Templates := "SrcType := Real" } EQ_Contact(in1 := "PLC_DATA".SMC_SILO_AG5, in2 := "C#7_RD_RUN".SMX_AG1)
      { S7_Templates := "SrcType := Real" } LT_Contact(in1 := "PLC_DATA".SMC_SILO_AG5, in2 := "C#7_RD_RUN".SMT)
   END_RUNG wire#w6
   RUNG wire#powerrail
      Contact( "C#2_WB"."NN_CAN AG5" )
   END_RUNG wire#w7
   RUNG wire#powerrail
      Contact( "XA_HET_AGG" )
   END_RUNG wire#w7
   RUNG wire#powerrail
      Contact( "C#2_WB".F2_SW_PAU )
   END_RUNG wire#w8
   RUNG wire#powerrail
      Contact( "C#2_WB".SW_PA_AG5 )
   END_RUNG wire#w8
   RUNG wire#powerrail
      { S7_Templates := "SrcType := Real" } EQ_Contact(in1 := "C#6_WD_CALIB".XUNG_AG1, in2 := 32767.0)
   END_RUNG wire#w8
   RUNG wire#powerrail
      P_Contact(operand := "PLC_BIT".AGG5_FU, bit := "P_AGG5_FU")
      wire#w9
      I_Contact( "C#1_RB"."XA W_AG1" )
      { S7_Templates := "SrcType := Real" } NE_Contact(in1 := "C#4_WD_WEIGHT".SV_AG5, in2 := 0.0)
      { S7_Templates := "SrcType := Real" } EQ_Contact(in1 := "PLC_DATA".SMC_SILO_AG5, in2 := "C#7_RD_RUN".SMX_AG1)
      Add(in1 := "PLC_DATA".SMC_SILO_AG5, in2 := 1.0, out => "PLC_DATA".SMC_SILO_AG5)
   END_RUNG
   RUNG wire#powerrail
      Contact( "P_RUN" )
      Contact( "PLC_BIT".AGG5_FU )
   END_RUNG wire#w9
   RUNG wire#powerrail
      Contact( "7.1.AGG5".STA_RUN )
      Coil( "C#1_RB".TTC_AG5 )
   END_RUNG
   // the same network as SCL:
   "9.1.DLC_AGG5"(ON := "PLC_BIT".RUN AND NOT "PLC_BIT".AGG5_FU AND NOT "C#1_RB"."XA W_AG1" AND (("PLC_BIT".AGG1_FU AND ("PLC_DATA".SMC_SILO_AG1 > "PLC_DATA".SMC_SILO_AG5)) OR ("C#4_WD_WEIGHT".SV_AG1 = 0.0)) AND (("PLC_BIT".AGG2_FU AND ("PLC_DATA".SMC_SILO_AG2 > "PLC_DATA".SMC_SILO_AG5)) OR ("C#4_WD_WEIGHT".SV_AG2 = 0.0)) AND (("PLC_BIT".AGG3_FU AND ("PLC_DATA".SMC_SILO_AG3 > "PLC_DATA".SMC_SILO_AG5)) OR ("C#4_WD_WEIGHT".SV_AG3 = 0.0)) AND (("PLC_BIT".AGG4_FU AND ("PLC_DATA".SMC_SILO_AG4 > "PLC_DATA".SMC_SILO_AG5)) OR ("C#4_WD_WEIGHT".SV_AG4 = 0.0)),   // "9.TIMER_DELAY"
                  CLOCK_1S := "Clock_10Hz",
                  T_DELAY := "C#4_WD_WEIGHT"."W_AG1_TG.DLC",
                  OUT => "9.1.DLC_AGG4".OUT,
                  T_OUT => "9.1.DLC_AGG4".T_OUT);
   "7.1.AGG5"(AUT := ("C#4_WD_WEIGHT".SV_AG5 <> 0.0) AND "PLC_BIT".RUN AND "PLC_BIT".AUT AND "9.1.DLC_AGG5".OUT AND NOT "PLC_BIT".AGG5_FU AND ("PLC_DATA".SMC_SILO_AG5 = "C#7_RD_RUN".SMX_AG1) AND ("PLC_DATA".SMC_SILO_AG5 < "C#7_RD_RUN".SMT),   // "7.WEIGHT_PROCESS"
              MAN1 := "C#2_WB"."NN_CAN AG5" OR "XA_HET_AGG",
              FAU := "C#2_WB".F2_SW_PAU OR "C#2_WB".SW_PA_AG5 OR ("C#6_WD_CALIB".XUNG_AG1 = 32767.0),
              FU_IN := "C#2_WB".NN_FU_AG5,
              X_CLOCK := "Clock_10Hz",
              EMTY_IN := "PLC_BIT".WAG1_EM,
              XNC_AUT := true,
              SV_IN := "C#4_WD_WEIGHT".SV_AG5,
              W_IN := "6.1.WAGG1".W_OUT5,
              W_RTD := "C#3_WD_SILO".AG5_KL_RTD,
              W_TR := "C#3_WD_SILO".AG5_SS_TREN,
              W_DU := "C#3_WD_SILO".AG5_SS_DUOI,
              T_ON := "C#3_WD_SILO".AG5_TG_ON_CAN,
              T_OFF := "C#3_WD_SILO".AG5_TG_OFF_CAN,
              T_DL := "C#3_WD_SILO".AG5_TG_ODC,
              PV_OUT => "C#7_RD_RUN".PV_AG5,
              PVM_OUT => "C#7_RD_RUN".PVM_AG5,
              FU_OUT => "PLC_BIT".AGG5_FU,
              Q_OUT1 => "C#1_RB"."CAN AG5",
              STA_RUN => "7.1.AGG5".STA_RUN);
   #_w1 := "PLC_BIT".AGG5_FU AND NOT "P_AGG5_FU";   // rising edge of "PLC_BIT".AGG5_FU
   "P_AGG5_FU" := "PLC_BIT".AGG5_FU;
   IF (#_w1 OR ("P_RUN" AND "PLC_BIT".AGG5_FU)) AND NOT "C#1_RB"."XA W_AG1" AND ("C#4_WD_WEIGHT".SV_AG5 <> 0.0) AND ("PLC_DATA".SMC_SILO_AG5 = "C#7_RD_RUN".SMX_AG1) THEN
       "PLC_DATA".SMC_SILO_AG5 := "PLC_DATA".SMC_SILO_AG5 + 1.0;
   END_IF;
   "C#1_RB".TTC_AG5 := "7.1.AGG5".STA_RUN;
END_REGION
END_FUNCTION
